FUNCTION_BLOCK DALI_TK_SR07
VAR_INPUT
	ID : DWORD;
END_VAR
VAR_OUTPUT
	Temp : UINT; (*Valore * 10 - 10,0°C => 100*)
END_VAR
VAR
	READ: FB_Rec_Generic;
	temperatura: DINT;
END_VAR

READ(
	str_KL6581:=enocean_buffer , 
	byNode:=1 , 
	dw_ID:=ID , 
	ar_Value=> , 
	by_Node=> , 
	by_STATE=> , 
	bReceive=> , 
	EnOceanTyp=> );
temperatura:=TRUNC((255-read.ar_Value[1])/0.6375);	
temp:=DINT_TO_UINT (temperatura);

END_FUNCTION_BLOCK

(* stored: Version 1.1.0.1, ProductVersion 3.1.4022.18
   POU DALI_TK_SR07: Id {4c16401b-44a3-4bce-be3e-79d380d27df3}, SpecialFunc None *)
